// TIA Portal V19 export
FUNCTION "PULSE VALVES" : Void   // FC21, STL
TITLE = PULSE VALVES
{ S7_Optimized_Access := 'TRUE' }
NAME : PULSEVAL
VERSION : 0.0
// Comment
// stored: AutoNumber false
BEGIN

NETWORK
TITLE = PULSE VALVES
// Comment
      AN    "PULSE 01.18 PRESTERILI";
      R     "T 46 PAUSE 01.13 PRES";
      R     "T 47 OPEN 01.13 PRES";
      JC    END;
      L     "MeasuredValues".TT0176REAL;  //"DB-ANALOG INPUT".TT0176MEAS
      L     "Setpoints".StaPulseY0113;  //"DB SETPOINTS".StaPulseY0113
      <R;
      JC    M001;
      A     "T 46 PAUSE 01.13 PRES";
      O     "T 47 OPEN 01.13 PRES";
      JC    M002;
      A     "MY0118";
      JC    M003;
      S     "MY0118";
      S     "TIM47";
      JU    M002;
M003: R     "MY0118";
      S     "TIM46";
      JU    M002;
M001: L     "MeasuredValues".TT0176REAL;  // "DB-ANALOG INPUT".TT0176MEAS
      L     "Setpoints".OpenY0113AtLowTemp;  // "DB SETPOINTS".OpenY0113AtLowTemp
      >R;
      JC    M002;
      S     "MY0118";
      R     "T 46 PAUSE 01.13 PRES";
      R     "T 47 OPEN 01.13 PRES";
M002: BEU;
END:  NOP   0;

NETWORK
TITLE = 
// Comment
      AN    "PULSE 01.13 CIP";
      JC    c001;
      A     "T 48 OPEN 01.13 CIP";
      JC    c001;
      A     "MY0113";
      JC    c002;
      S     "MY0113";
      R     "PULSE 01.13 CIP";
      JU    c001;
c002: R     "MY0113";
      S     "TIM48";
c001: NOP   0;

NETWORK
TITLE = 
// Comment
      AN    "PULSE 01.08 CIP";
      R     "T 49 OPEN 01.08 CIP";
      R     "T 50 OPEN 01.24 CIP";
      R     "T 51 PAUSE 01.08 CIP";
      JC    c003;
      AN    "UHT_STERILE?";
      JC    c004;
      R     "MY0108";
      R     "MY0124";
      R     "MY0144";
      JU    c003;
c004: A     "T 51 PAUSE 01.08 CIP";
      JC    c003;
      AN    "T 49 OPEN 01.08 CIP";
      JC    c005;
      A     "T 50 OPEN 01.24 CIP";
      JC    c003;
      R     "MY0124";
      R     "MY0144";
      JU    c003;
c005: A     "MY0108";
      JC    c006;
      S     "MY0108";
      S     "TIM49";
      S     "MY0124";
      S     "TIM50";
      S     "MY0144";
      JU    c003;
//M003:
c006: R     "MY0108";
      S     "TIM51";
      R     "MY0124";
c003: NOP   0;
END_FUNCTION
